{attribute 'qualified_only'}
{attribute 'strict'}
TYPE E_NappienNumerointi :
(
	Vipu1,
	Vipu2,
	Nappi1
);
END_TYPE

(* stored: Version 1.1.0.1, ProductVersion 3.1.4024.10
   DUT E_NappienNumerointi: Id {317754fe-34bc-4148-abf0-4f663ed440cf} *)
